FUNCTION_BLOCK FB_TempLogging_OpcUa
VAR
  // used data
  _pAdsPh  : ARRAY[1..nC_MaxPHs] OF POINTER TO ST_ADS_PH;
  _nRegPhs : UDINT;                                           (*number o registered printheads*)

  // timing
  fb_TonMaxTemp                             : TON;            (*Timer for max temperature*)
  tL_TimeMaxTemp                            : TIME := T#10S;  (*Interval for max temperature*)
  i                                         : UDINT;
  
  {attribute 'OPC.UA.DA':='1'}
  iL_TempActValuePH                         : ARRAY[1..nC_MaxPHs] OF INT;       (*Actual temperature PHx*)
  {attribute 'OPC.UA.DA':='1'}
  iL_TempMaxValuePH                         : ARRAY[1..nC_MaxPHs] OF INT;       (*Max temperature in interval PHx*)
END_VAR
VAR CONSTANT
  nC_MaxPHs                                 : UDINT := 8;
END_VAR

(*Detect max temp value in defined interval*)
fb_TonMaxTemp(IN := NOT fb_TonMaxTemp.Q, PT := tL_TimeMaxTemp);
IF fb_TonMaxTemp.Q THEN
  
  FOR i:=1 TO _nRegPhs DO 
    iL_TempActValuePH[i] := iL_TempMaxValuePH[i];
    iL_TempMaxValuePH[i] := _pAdsPh[i]^.iO_Temperature;
	END_FOR

END_IF

iL_TempMaxValuePH[i] := MAX(iL_TempMaxValuePH[i], _pAdsPh[i]^.iO_Temperature);

METHOD registerPH : BOOL
VAR_INPUT
  pAdsPh : POINTER TO ST_ADS_PH;
END_VAR
IF pAdsPh = 0 THEN RETURN; END_IF 
IF _nRegPhs >= nC_MaxPHs THEN F_LogError('Too many phs already registered'); RETURN; END_IF 


_nRegPhs := _nRegPhs + 1;
_pAdsPh[_nRegPhs] := pAdsPh;
END_METHOD

END_FUNCTION_BLOCK

(* stored: Version 1.1.0.1, ProductVersion 3.1.4024.11
   POU FB_TempLogging_OpcUa: Id {fd731e1d-6860-4dd7-8b04-05f2e3a3a0fe}, SpecialFunc None
   Method registerPH: Id {5b53e921-ab1c-4caf-b430-fc1a5c280839} *)
